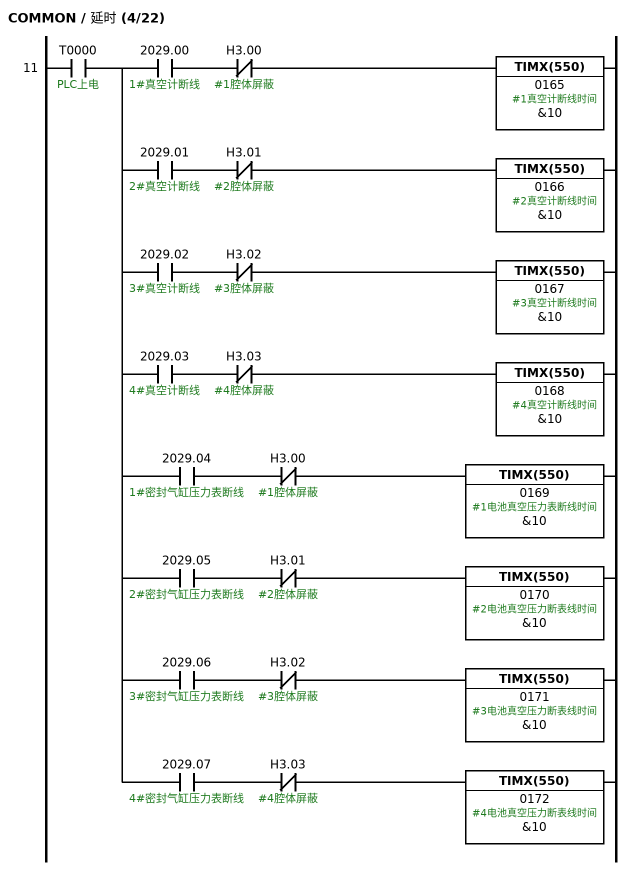
; [picture p384: COMMON / 延时, rungs 11-11]
; rung 11
LD T0000  ; PLC上电
OUT TR0
AND 2029.00  ; 1#真空计断线
ANDNOT H3.00  ; #1腔体屏蔽
TIMX(550) 0165 &10  ; #1真空计断线时间
LD TR0
AND 2029.01  ; 2#真空计断线
ANDNOT H3.01  ; #2腔体屏蔽
TIMX(550) 0166 &10  ; #2真空计断线时间
LD TR0
AND 2029.02  ; 3#真空计断线
ANDNOT H3.02  ; #3腔体屏蔽
TIMX(550) 0167 &10  ; #3真空计断线时间
LD TR0
AND 2029.03  ; 4#真空计断线
ANDNOT H3.03  ; #4腔体屏蔽
TIMX(550) 0168 &10  ; #4真空计断线时间
LD TR0
AND 2029.04  ; 1#密封气缸压力表断线
ANDNOT H3.00  ; #1腔体屏蔽
TIMX(550) 0169 &10  ; #1电池真空压力表断线时间
LD TR0
AND 2029.05  ; 2#密封气缸压力表断线
ANDNOT H3.01  ; #2腔体屏蔽
TIMX(550) 0170 &10  ; #2电池真空压力断表线时间
LD TR0
AND 2029.06  ; 3#密封气缸压力表断线
ANDNOT H3.02  ; #3腔体屏蔽
TIMX(550) 0171 &10  ; #3电池真空压力断表线时间
LD TR0
AND 2029.07  ; 4#密封气缸压力表断线
ANDNOT H3.03  ; #4腔体屏蔽
TIMX(550) 0172 &10  ; #4电池真空压力断表线时间

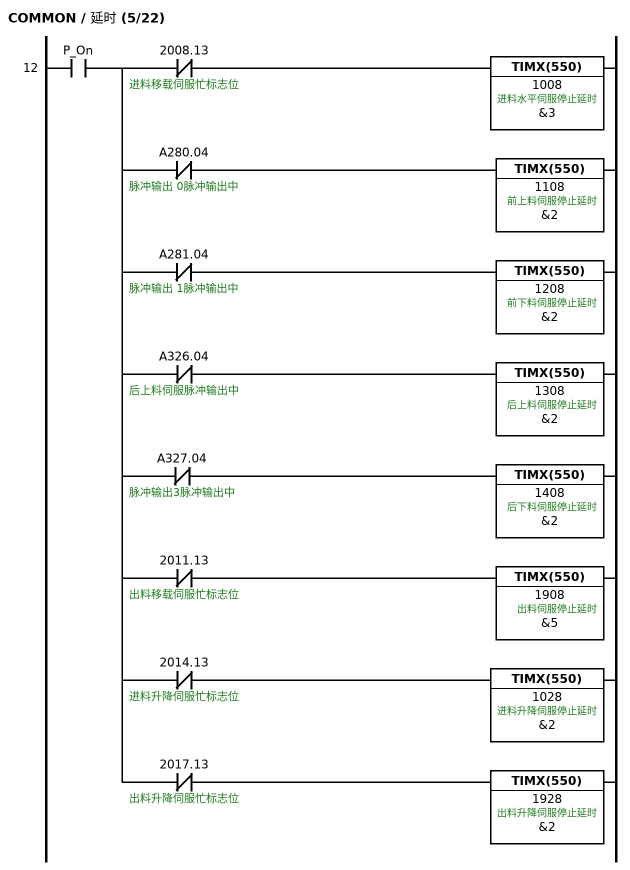
; rung 12
LD P_On
OUT TR0
ANDNOT 2008.13  ; 进料移载伺服忙标志位
TIMX(550) 1008 &3  ; 进料水平伺服停止延时
LD TR0
ANDNOT A280.04  ; 脉冲输出 0脉冲输出中
TIMX(550) 1108 &2  ; 前上料伺服停止延时
LD TR0
ANDNOT A281.04  ; 脉冲输出 1脉冲输出中
TIMX(550) 1208 &2  ; 前下料伺服停止延时
LD TR0
ANDNOT A326.04  ; 后上料伺服脉冲输出中
TIMX(550) 1308 &2  ; 后上料伺服停止延时
LD TR0
ANDNOT A327.04  ; 脉冲输出3脉冲输出中
TIMX(550) 1408 &2  ; 后下料伺服停止延时
LD TR0
ANDNOT 2011.13  ; 出料移载伺服忙标志位
TIMX(550) 1908 &5  ; 出料伺服停止延时
LD TR0
ANDNOT 2014.13  ; 进料升降伺服忙标志位
TIMX(550) 1028 &2  ; 进料升降伺服停止延时
LD TR0
ANDNOT 2017.13  ; 出料升降伺服忙标志位
TIMX(550) 1928 &2  ; 出料升降伺服停止延时

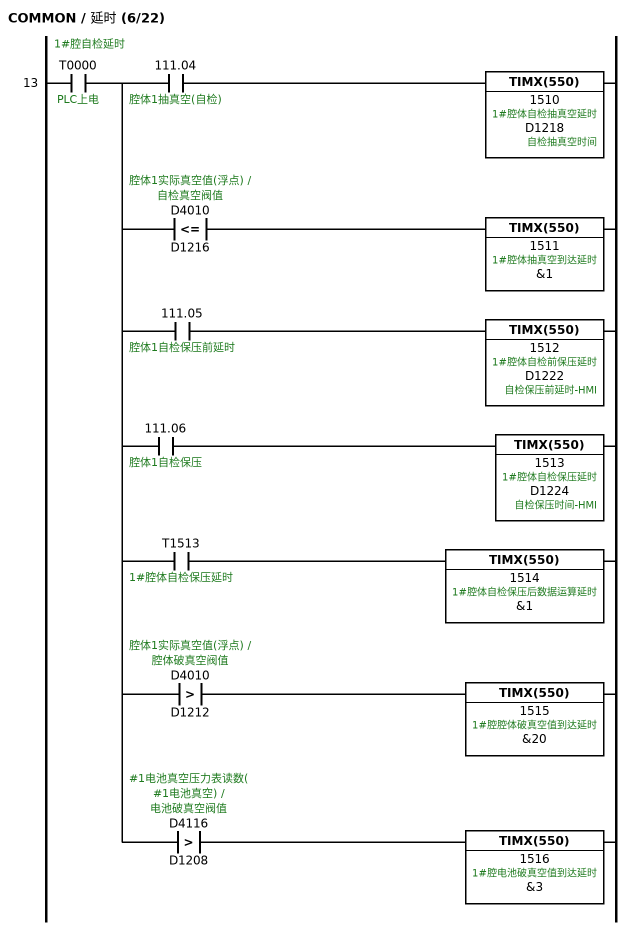
; rung 13: 1#腔自检延时
LD T0000  ; PLC上电
OUT TR0
AND 111.04  ; 腔体1抽真空(自检)
TIMX(550) 1510 D1218  ; 自检抽真空时间, 1#腔体自检抽真空延时
LD TR0
AND<=F(332) D4010 D1216  ; 腔体1实际真空值(浮点), 自检真空阀值
TIMX(550) 1511 &1  ; 1#腔体抽真空到达延时
LD TR0
AND 111.05  ; 腔体1自检保压前延时
TIMX(550) 1512 D1222  ; 自检保压前延时-HMI, 1#腔体自检前保压延时
LD TR0
AND 111.06  ; 腔体1自检保压
TIMX(550) 1513 D1224  ; 自检保压时间-HMI, 1#腔体自检保压延时
LD TR0
AND T1513  ; 1#腔体自检保压延时
TIMX(550) 1514 &1  ; 1#腔体自检保压后数据运算延时
LD TR0
AND>F(333) D4010 D1212  ; 腔体1实际真空值(浮点), 腔体破真空阀值
TIMX(550) 1515 &20  ; 1#腔腔体破真空值到达延时
LD TR0
AND>F(333) D4116 D1208  ; #1电池真空压力表读数(#1电池真空), 电池破真空阀值
TIMX(550) 1516 &3  ; 1#腔电池破真空值到达延时

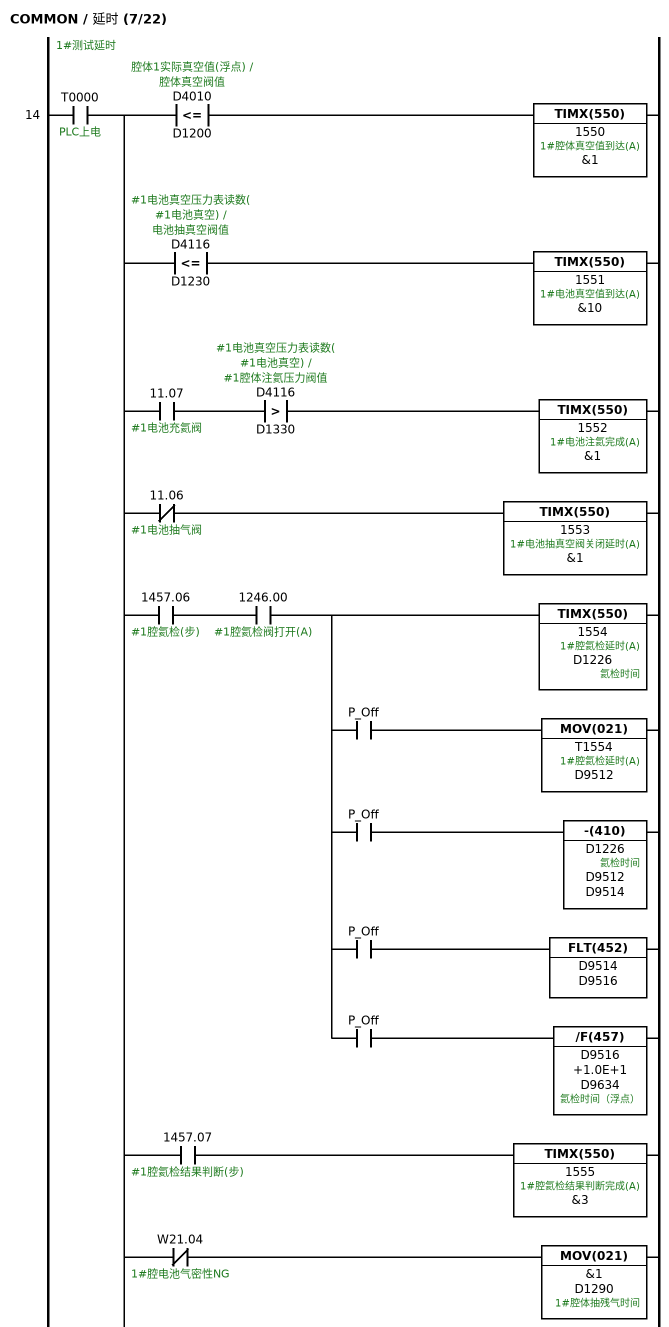

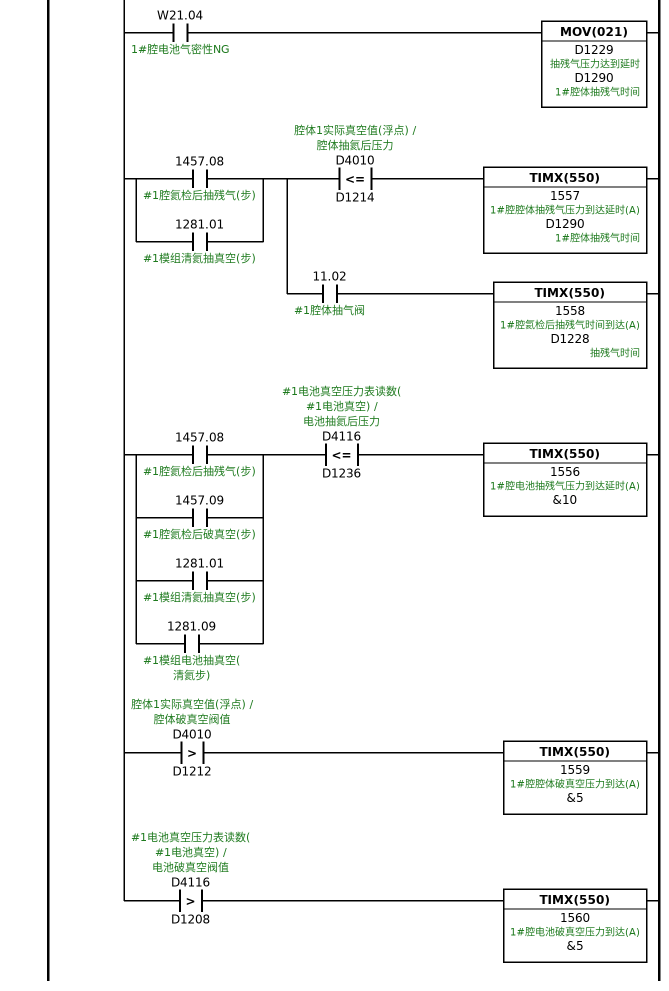
; rung 14: 1#测试延时
LD T0000  ; PLC上电
OUT TR0
AND<=F(332) D4010 D1200  ; 腔体1实际真空值(浮点), 腔体真空阀值
TIMX(550) 1550 &1  ; 1#腔体真空值到达(A)
LD TR0
AND<=F(332) D4116 D1230  ; #1电池真空压力表读数(#1电池真空), 电池抽真空阀值
TIMX(550) 1551 &10  ; 1#电池真空值到达(A)
LD TR0
AND 11.07  ; #1电池充氦阀
AND>F(333) D4116 D1330  ; #1电池真空压力表读数(#1电池真空), #1腔体注氦压力阀值
TIMX(550) 1552 &1  ; 1#电池注氦完成(A)
LD TR0
ANDNOT 11.06  ; #1电池抽气阀
TIMX(550) 1553 &1  ; 1#电池抽真空阀关闭延时(A)
LD TR0
AND 1457.06  ; #1腔氦检(步)
AND 1246.00  ; #1腔氦检阀打开(A)
OUT TR1
TIMX(550) 1554 D1226  ; 氦检时间, 1#腔氦检延时(A)
AND P_Off
MOV(021) T1554 D9512  ; 1#腔氦检延时(A)
LD TR1
AND P_Off
-(410) D1226 D9512 D9514  ; 氦检时间
LD TR1
AND P_Off
FLT(452) D9514 D9516
LD TR1
AND P_Off
/F(457) D9516 +1.0E+1 D9634  ; 氦检时间（浮点）
LD TR0
AND 1457.07  ; #1腔氦检结果判断(步)
TIMX(550) 1555 &3  ; 1#腔氦检结果判断完成(A)
LD TR0
ANDNOT W21.04  ; 1#腔电池气密性NG
MOV(021) &1 D1290  ; 1#腔体抽残气时间
LD TR0
AND W21.04  ; 1#腔电池气密性NG
MOV(021) D1229 D1290  ; 抽残气压力达到延时, 1#腔体抽残气时间
LD TR0
LD 1457.08  ; #1腔氦检后抽残气(步)
OR 1281.01  ; #1模组清氦抽真空(步)
ANDLD
OUT TR1
AND<=F(332) D4010 D1214  ; 腔体1实际真空值(浮点), 腔体抽氦后压力
TIMX(550) 1557 D1290  ; 1#腔体抽残气时间, 1#腔腔体抽残气压力到达延时(A)
LD TR1
AND 11.02  ; #1腔体抽气阀
TIMX(550) 1558 D1228  ; 抽残气时间, 1#腔氦检后抽残气时间到达(A)
LD TR0
LD 1457.08  ; #1腔氦检后抽残气(步)
OR 1457.09  ; #1腔氦检后破真空(步)
OR 1281.01  ; #1模组清氦抽真空(步)
OR 1281.09  ; #1模组电池抽真空(清氦步)
ANDLD
AND<=F(332) D4116 D1236  ; #1电池真空压力表读数(#1电池真空), 电池抽氦后压力
TIMX(550) 1556 &10  ; 1#腔电池抽残气压力到达延时(A)
LD TR0
AND>F(333) D4010 D1212  ; 腔体1实际真空值(浮点), 腔体破真空阀值
TIMX(550) 1559 &5  ; 1#腔腔体破真空压力到达(A)
LD TR0
AND>F(333) D4116 D1208  ; #1电池真空压力表读数(#1电池真空), 电池破真空阀值
TIMX(550) 1560 &5  ; 1#腔电池破真空压力到达(A)

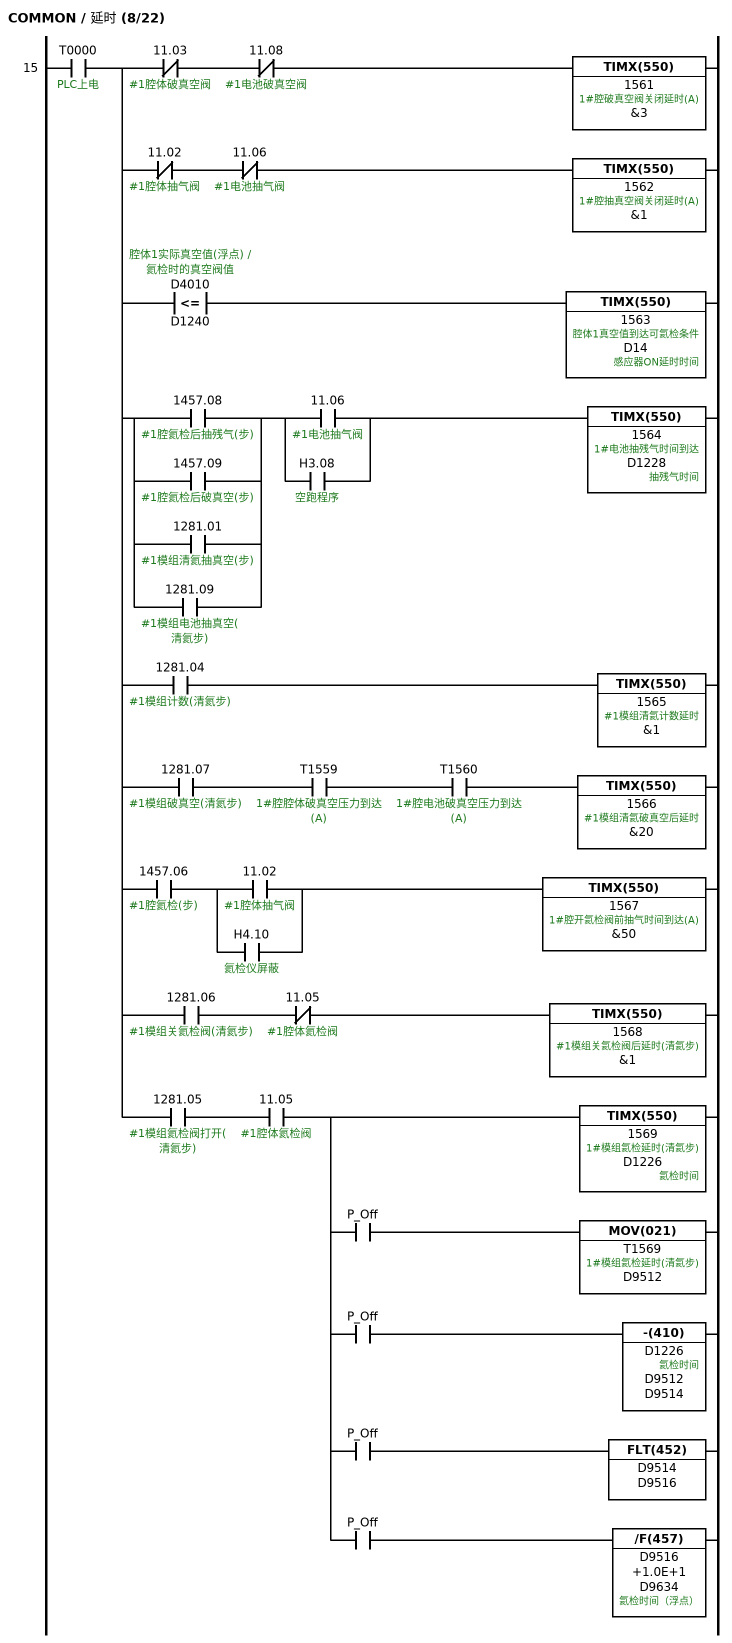
; rung 15
LD T0000  ; PLC上电
OUT TR0
ANDNOT 11.03  ; #1腔体破真空阀
ANDNOT 11.08  ; #1电池破真空阀
TIMX(550) 1561 &3  ; 1#腔破真空阀关闭延时(A)
LD TR0
ANDNOT 11.02  ; #1腔体抽气阀
ANDNOT 11.06  ; #1电池抽气阀
TIMX(550) 1562 &1  ; 1#腔抽真空阀关闭延时(A)
LD TR0
AND<=F(332) D4010 D1240  ; 腔体1实际真空值(浮点), 氦检时的真空阀值
TIMX(550) 1563 D14  ; 感应器ON延时时间, 腔体1真空值到达可氦检条件
LD TR0
LD 1457.08  ; #1腔氦检后抽残气(步)
OR 1457.09  ; #1腔氦检后破真空(步)
OR 1281.01  ; #1模组清氦抽真空(步)
OR 1281.09  ; #1模组电池抽真空(清氦步)
ANDLD
LD 11.06  ; #1电池抽气阀
OR H3.08  ; 空跑程序
ANDLD
TIMX(550) 1564 D1228  ; 抽残气时间, 1#电池抽残气时间到达
LD TR0
AND 1281.04  ; #1模组计数(清氦步)
TIMX(550) 1565 &1  ; #1模组清氦计数延时
LD TR0
AND 1281.07  ; #1模组破真空(清氦步)
AND T1559  ; 1#腔腔体破真空压力到达(A)
AND T1560  ; 1#腔电池破真空压力到达(A)
TIMX(550) 1566 &20  ; #1模组清氦破真空后延时
LD TR0
AND 1457.06  ; #1腔氦检(步)
LD 11.02  ; #1腔体抽气阀
OR H4.10  ; 氦检仪屏蔽
ANDLD
TIMX(550) 1567 &50  ; 1#腔开氦检阀前抽气时间到达(A)
LD TR0
AND 1281.06  ; #1模组关氦检阀(清氦步)
ANDNOT 11.05  ; #1腔体氦检阀
TIMX(550) 1568 &1  ; #1模组关氦检阀后延时(清氦步)
LD TR0
AND 1281.05  ; #1模组氦检阀打开(清氦步)
AND 11.05  ; #1腔体氦检阀
OUT TR0
TIMX(550) 1569 D1226  ; 氦检时间, 1#模组氦检延时(清氦步)
AND P_Off
MOV(021) T1569 D9512  ; 1#模组氦检延时(清氦步)
LD TR0
AND P_Off
-(410) D1226 D9512 D9514  ; 氦检时间
LD TR0
AND P_Off
FLT(452) D9514 D9516
LD TR0
AND P_Off
/F(457) D9516 +1.0E+1 D9634  ; 氦检时间（浮点）

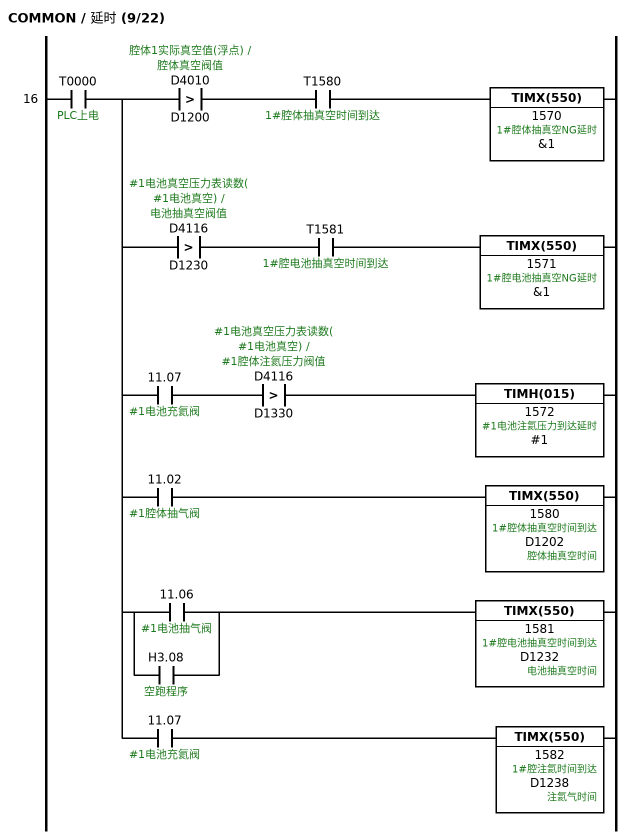
; rung 16
LD T0000  ; PLC上电
OUT TR0
AND>F(333) D4010 D1200  ; 腔体1实际真空值(浮点), 腔体真空阀值
AND T1580  ; 1#腔体抽真空时间到达
TIMX(550) 1570 &1  ; 1#腔体抽真空NG延时
LD TR0
AND>F(333) D4116 D1230  ; #1电池真空压力表读数(#1电池真空), 电池抽真空阀值
AND T1581  ; 1#腔电池抽真空时间到达
TIMX(550) 1571 &1  ; 1#腔电池抽真空NG延时
LD TR0
AND 11.07  ; #1电池充氦阀
AND>F(333) D4116 D1330  ; #1电池真空压力表读数(#1电池真空), #1腔体注氦压力阀值
TIMH(015) 1572 #1  ; #1电池注氦压力到达延时
LD TR0
AND 11.02  ; #1腔体抽气阀
TIMX(550) 1580 D1202  ; 腔体抽真空时间, 1#腔体抽真空时间到达
LD TR0
LD 11.06  ; #1电池抽气阀
OR H3.08  ; 空跑程序
ANDLD
TIMX(550) 1581 D1232  ; 电池抽真空时间, 1#腔电池抽真空时间到达
LD TR0
AND 11.07  ; #1电池充氦阀
TIMX(550) 1582 D1238  ; 注氦气时间, 1#腔注氦时间到达

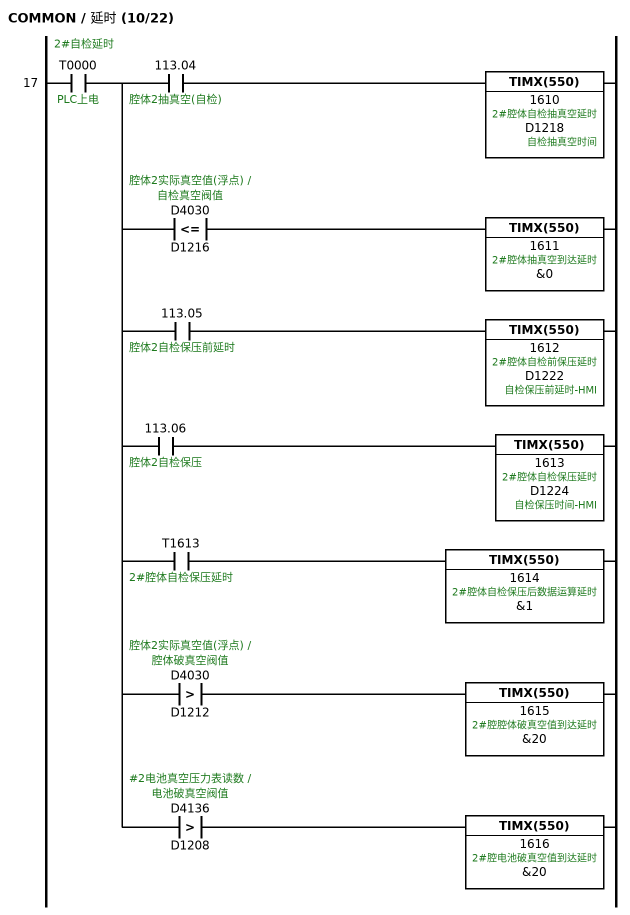
; rung 17: 2#自检延时
LD T0000  ; PLC上电
OUT TR0
AND 113.04  ; 腔体2抽真空(自检)
TIMX(550) 1610 D1218  ; 自检抽真空时间, 2#腔体自检抽真空延时
LD TR0
AND<=F(332) D4030 D1216  ; 腔体2实际真空值(浮点), 自检真空阀值
TIMX(550) 1611 &0  ; 2#腔体抽真空到达延时
LD TR0
AND 113.05  ; 腔体2自检保压前延时
TIMX(550) 1612 D1222  ; 自检保压前延时-HMI, 2#腔体自检前保压延时
LD TR0
AND 113.06  ; 腔体2自检保压
TIMX(550) 1613 D1224  ; 自检保压时间-HMI, 2#腔体自检保压延时
LD TR0
AND T1613  ; 2#腔体自检保压延时
TIMX(550) 1614 &1  ; 2#腔体自检保压后数据运算延时
LD TR0
AND>F(333) D4030 D1212  ; 腔体2实际真空值(浮点), 腔体破真空阀值
TIMX(550) 1615 &20  ; 2#腔腔体破真空值到达延时
LD TR0
AND>F(333) D4136 D1208  ; #2电池真空压力表读数, 电池破真空阀值
TIMX(550) 1616 &20  ; 2#腔电池破真空值到达延时

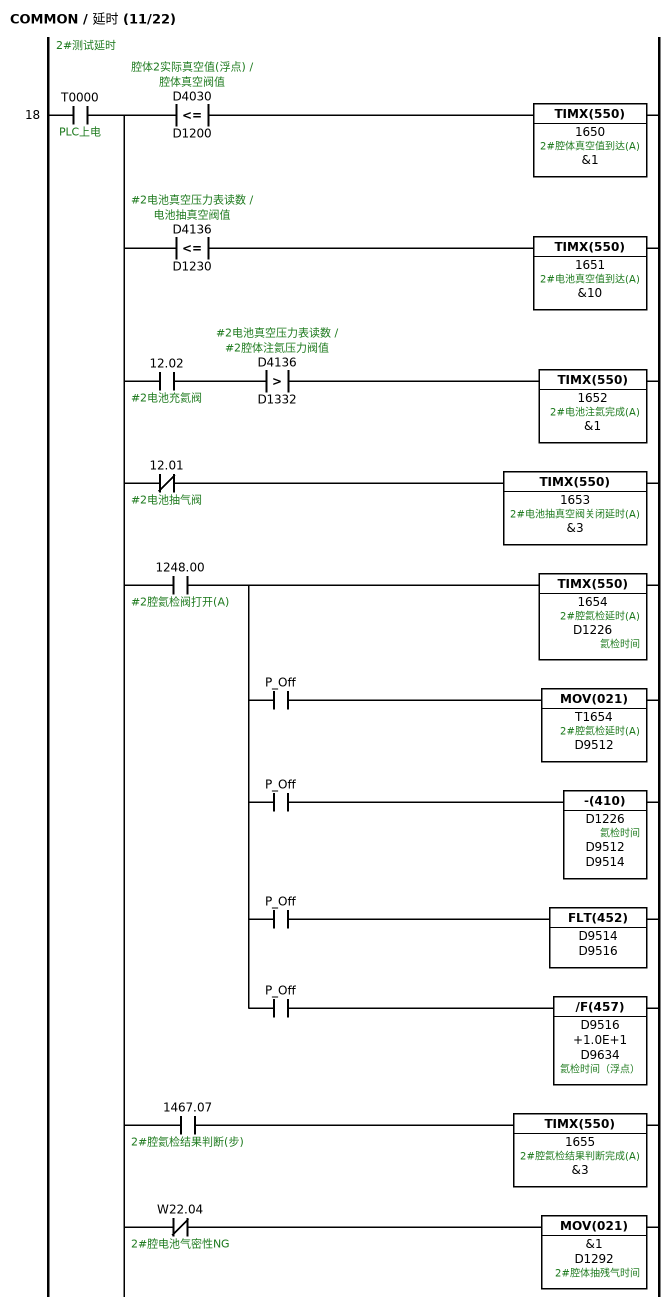

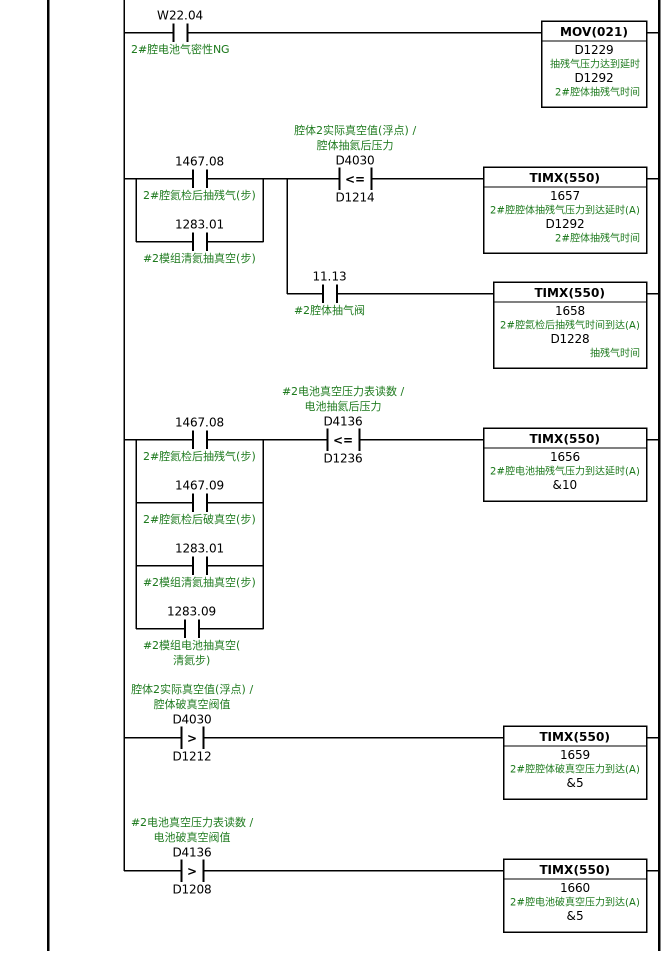
; rung 18: 2#测试延时
LD T0000  ; PLC上电
OUT TR0
AND<=F(332) D4030 D1200  ; 腔体2实际真空值(浮点), 腔体真空阀值
TIMX(550) 1650 &1  ; 2#腔体真空值到达(A)
LD TR0
AND<=F(332) D4136 D1230  ; #2电池真空压力表读数, 电池抽真空阀值
TIMX(550) 1651 &10  ; 2#电池真空值到达(A)
LD TR0
AND 12.02  ; #2电池充氦阀
AND>F(333) D4136 D1332  ; #2电池真空压力表读数, #2腔体注氦压力阀值
TIMX(550) 1652 &1  ; 2#电池注氦完成(A)
LD TR0
ANDNOT 12.01  ; #2电池抽气阀
TIMX(550) 1653 &3  ; 2#电池抽真空阀关闭延时(A)
LD TR0
AND 1248.00  ; #2腔氦检阀打开(A)
OUT TR1
TIMX(550) 1654 D1226  ; 氦检时间, 2#腔氦检延时(A)
AND P_Off
MOV(021) T1654 D9512  ; 2#腔氦检延时(A)
LD TR1
AND P_Off
-(410) D1226 D9512 D9514  ; 氦检时间
LD TR1
AND P_Off
FLT(452) D9514 D9516
LD TR1
AND P_Off
/F(457) D9516 +1.0E+1 D9634  ; 氦检时间（浮点）
LD TR0
AND 1467.07  ; 2#腔氦检结果判断(步)
TIMX(550) 1655 &3  ; 2#腔氦检结果判断完成(A)
LD TR0
ANDNOT W22.04  ; 2#腔电池气密性NG
MOV(021) &1 D1292  ; 2#腔体抽残气时间
LD TR0
AND W22.04  ; 2#腔电池气密性NG
MOV(021) D1229 D1292  ; 抽残气压力达到延时, 2#腔体抽残气时间
LD TR0
LD 1467.08  ; 2#腔氦检后抽残气(步)
OR 1283.01  ; #2模组清氦抽真空(步)
ANDLD
OUT TR1
AND<=F(332) D4030 D1214  ; 腔体2实际真空值(浮点), 腔体抽氦后压力
TIMX(550) 1657 D1292  ; 2#腔体抽残气时间, 2#腔腔体抽残气压力到达延时(A)
LD TR1
AND 11.13  ; #2腔体抽气阀
TIMX(550) 1658 D1228  ; 抽残气时间, 2#腔氦检后抽残气时间到达(A)
LD TR0
LD 1467.08  ; 2#腔氦检后抽残气(步)
OR 1467.09  ; 2#腔氦检后破真空(步)
OR 1283.01  ; #2模组清氦抽真空(步)
OR 1283.09  ; #2模组电池抽真空(清氦步)
ANDLD
AND<=F(332) D4136 D1236  ; #2电池真空压力表读数, 电池抽氦后压力
TIMX(550) 1656 &10  ; 2#腔电池抽残气压力到达延时(A)
LD TR0
AND>F(333) D4030 D1212  ; 腔体2实际真空值(浮点), 腔体破真空阀值
TIMX(550) 1659 &5  ; 2#腔腔体破真空压力到达(A)
LD TR0
AND>F(333) D4136 D1208  ; #2电池真空压力表读数, 电池破真空阀值
TIMX(550) 1660 &5  ; 2#腔电池破真空压力到达(A)

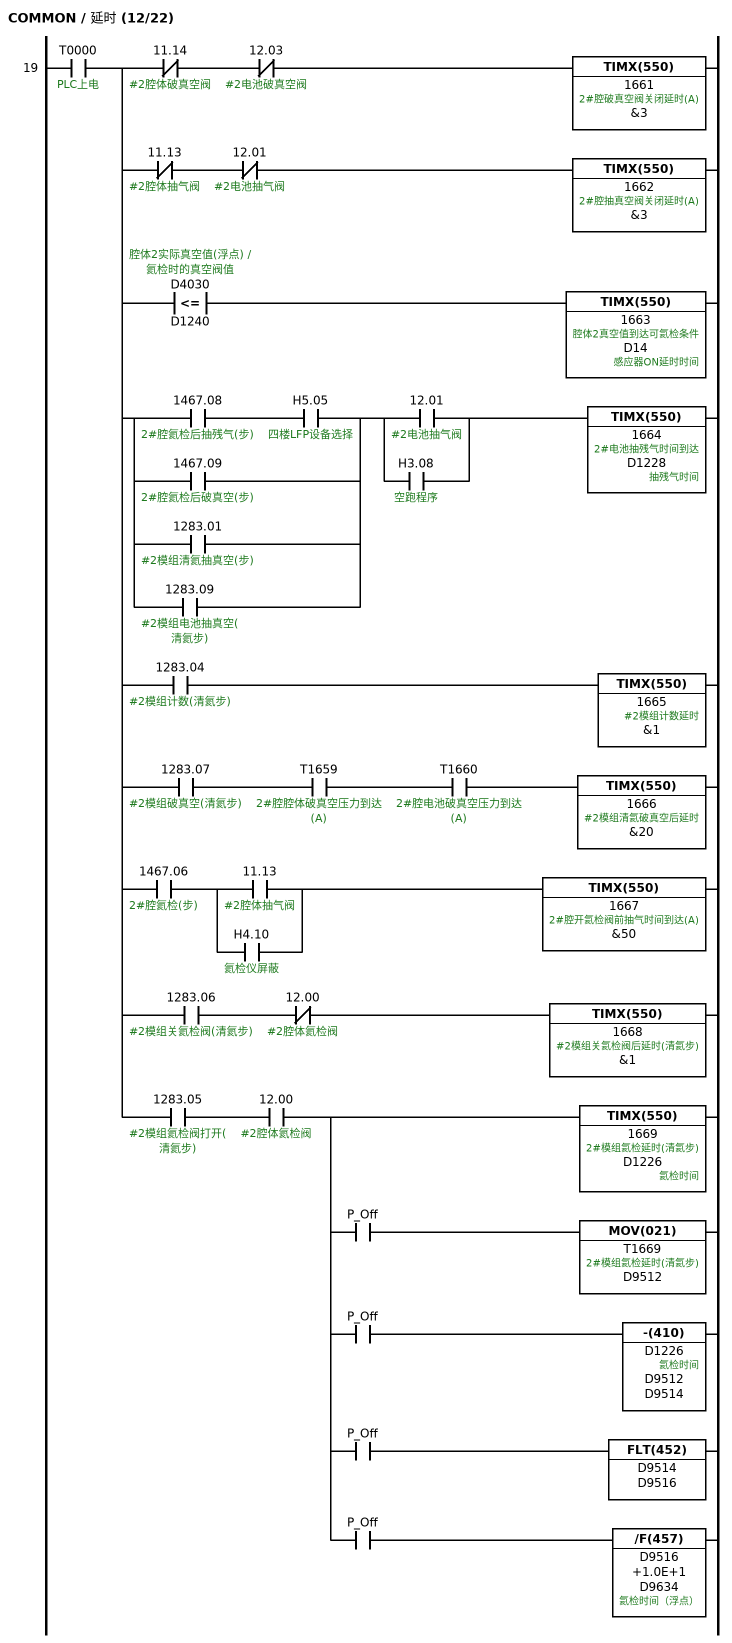
; rung 19
LD T0000  ; PLC上电
OUT TR0
ANDNOT 11.14  ; #2腔体破真空阀
ANDNOT 12.03  ; #2电池破真空阀
TIMX(550) 1661 &3  ; 2#腔破真空阀关闭延时(A)
LD TR0
ANDNOT 11.13  ; #2腔体抽气阀
ANDNOT 12.01  ; #2电池抽气阀
TIMX(550) 1662 &3  ; 2#腔抽真空阀关闭延时(A)
LD TR0
AND<=F(332) D4030 D1240  ; 腔体2实际真空值(浮点), 氦检时的真空阀值
TIMX(550) 1663 D14  ; 感应器ON延时时间, 腔体2真空值到达可氦检条件
LD TR0
LD 1467.08  ; 2#腔氦检后抽残气(步)
AND H5.05  ; 四楼LFP设备选择
OR 1467.09  ; 2#腔氦检后破真空(步)
OR 1283.01  ; #2模组清氦抽真空(步)
OR 1283.09  ; #2模组电池抽真空(清氦步)
ANDLD
LD 12.01  ; #2电池抽气阀
OR H3.08  ; 空跑程序
ANDLD
TIMX(550) 1664 D1228  ; 抽残气时间, 2#电池抽残气时间到达
LD TR0
AND 1283.04  ; #2模组计数(清氦步)
TIMX(550) 1665 &1  ; #2模组计数延时
LD TR0
AND 1283.07  ; #2模组破真空(清氦步)
AND T1659  ; 2#腔腔体破真空压力到达(A)
AND T1660  ; 2#腔电池破真空压力到达(A)
TIMX(550) 1666 &20  ; #2模组清氦破真空后延时
LD TR0
AND 1467.06  ; 2#腔氦检(步)
LD 11.13  ; #2腔体抽气阀
OR H4.10  ; 氦检仪屏蔽
ANDLD
TIMX(550) 1667 &50  ; 2#腔开氦检阀前抽气时间到达(A)
LD TR0
AND 1283.06  ; #2模组关氦检阀(清氦步)
ANDNOT 12.00  ; #2腔体氦检阀
TIMX(550) 1668 &1  ; #2模组关氦检阀后延时(清氦步)
LD TR0
AND 1283.05  ; #2模组氦检阀打开(清氦步)
AND 12.00  ; #2腔体氦检阀
OUT TR0
TIMX(550) 1669 D1226  ; 氦检时间, 2#模组氦检延时(清氦步)
AND P_Off
MOV(021) T1669 D9512  ; 2#模组氦检延时(清氦步)
LD TR0
AND P_Off
-(410) D1226 D9512 D9514  ; 氦检时间
LD TR0
AND P_Off
FLT(452) D9514 D9516
LD TR0
AND P_Off
/F(457) D9516 +1.0E+1 D9634  ; 氦检时间（浮点）

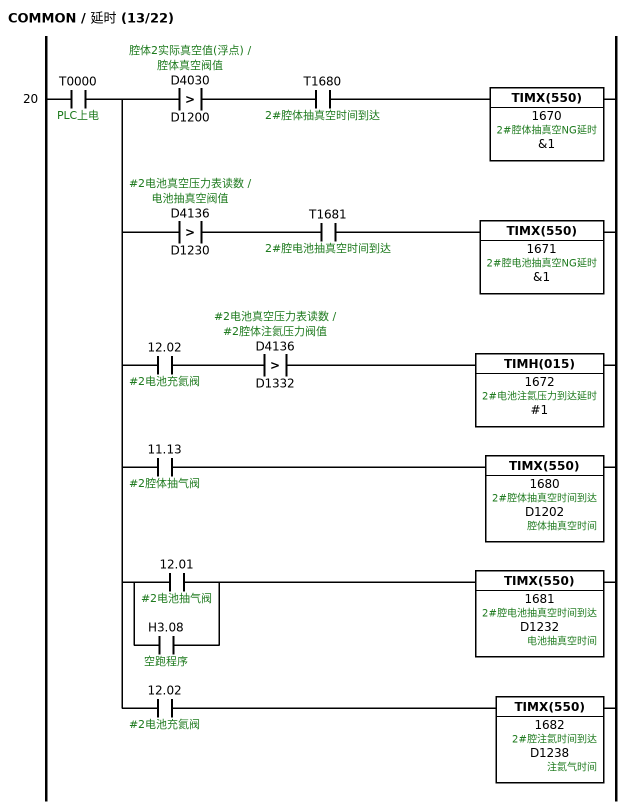
; rung 20
LD T0000  ; PLC上电
OUT TR0
AND>F(333) D4030 D1200  ; 腔体2实际真空值(浮点), 腔体真空阀值
AND T1680  ; 2#腔体抽真空时间到达
TIMX(550) 1670 &1  ; 2#腔体抽真空NG延时
LD TR0
AND>F(333) D4136 D1230  ; #2电池真空压力表读数, 电池抽真空阀值
AND T1681  ; 2#腔电池抽真空时间到达
TIMX(550) 1671 &1  ; 2#腔电池抽真空NG延时
LD TR0
AND 12.02  ; #2电池充氦阀
AND>F(333) D4136 D1332  ; #2电池真空压力表读数, #2腔体注氦压力阀值
TIMH(015) 1672 #1  ; 2#电池注氦压力到达延时
LD TR0
AND 11.13  ; #2腔体抽气阀
TIMX(550) 1680 D1202  ; 腔体抽真空时间, 2#腔体抽真空时间到达
LD TR0
LD 12.01  ; #2电池抽气阀
OR H3.08  ; 空跑程序
ANDLD
TIMX(550) 1681 D1232  ; 电池抽真空时间, 2#腔电池抽真空时间到达
LD TR0
AND 12.02  ; #2电池充氦阀
TIMX(550) 1682 D1238  ; 注氦气时间, 2#腔注氦时间到达

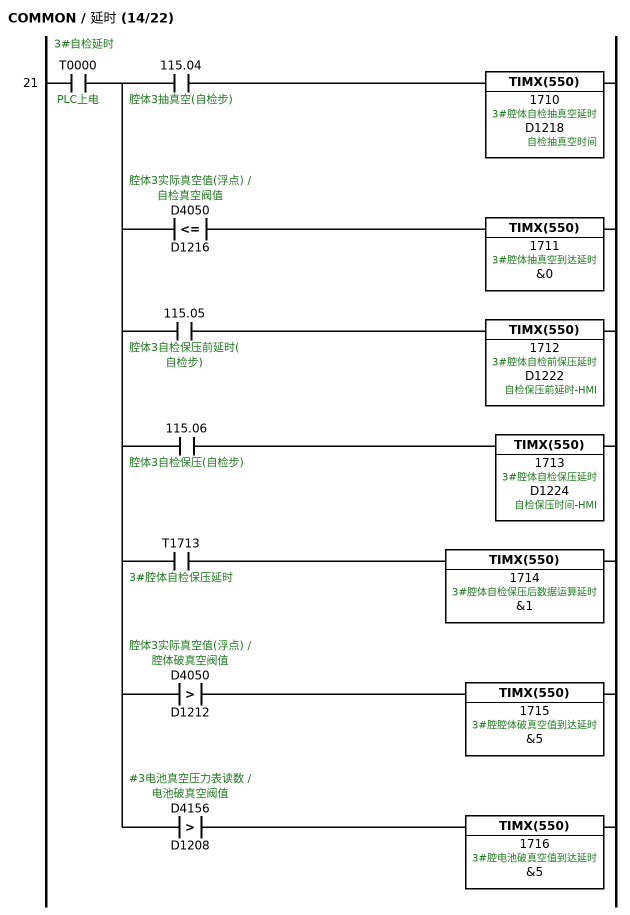
; rung 21: 3#自检延时
LD T0000  ; PLC上电
OUT TR0
AND 115.04  ; 腔体3抽真空(自检步)
TIMX(550) 1710 D1218  ; 自检抽真空时间, 3#腔体自检抽真空延时
LD TR0
AND<=F(332) D4050 D1216  ; 腔体3实际真空值(浮点), 自检真空阀值
TIMX(550) 1711 &0  ; 3#腔体抽真空到达延时
LD TR0
AND 115.05  ; 腔体3自检保压前延时(自检步)
TIMX(550) 1712 D1222  ; 自检保压前延时-HMI, 3#腔体自检前保压延时
LD TR0
AND 115.06  ; 腔体3自检保压(自检步)
TIMX(550) 1713 D1224  ; 自检保压时间-HMI, 3#腔体自检保压延时
LD TR0
AND T1713  ; 3#腔体自检保压延时
TIMX(550) 1714 &1  ; 3#腔体自检保压后数据运算延时
LD TR0
AND>F(333) D4050 D1212  ; 腔体3实际真空值(浮点), 腔体破真空阀值
TIMX(550) 1715 &5  ; 3#腔腔体破真空值到达延时
LD TR0
AND>F(333) D4156 D1208  ; #3电池真空压力表读数, 电池破真空阀值
TIMX(550) 1716 &5  ; 3#腔电池破真空值到达延时

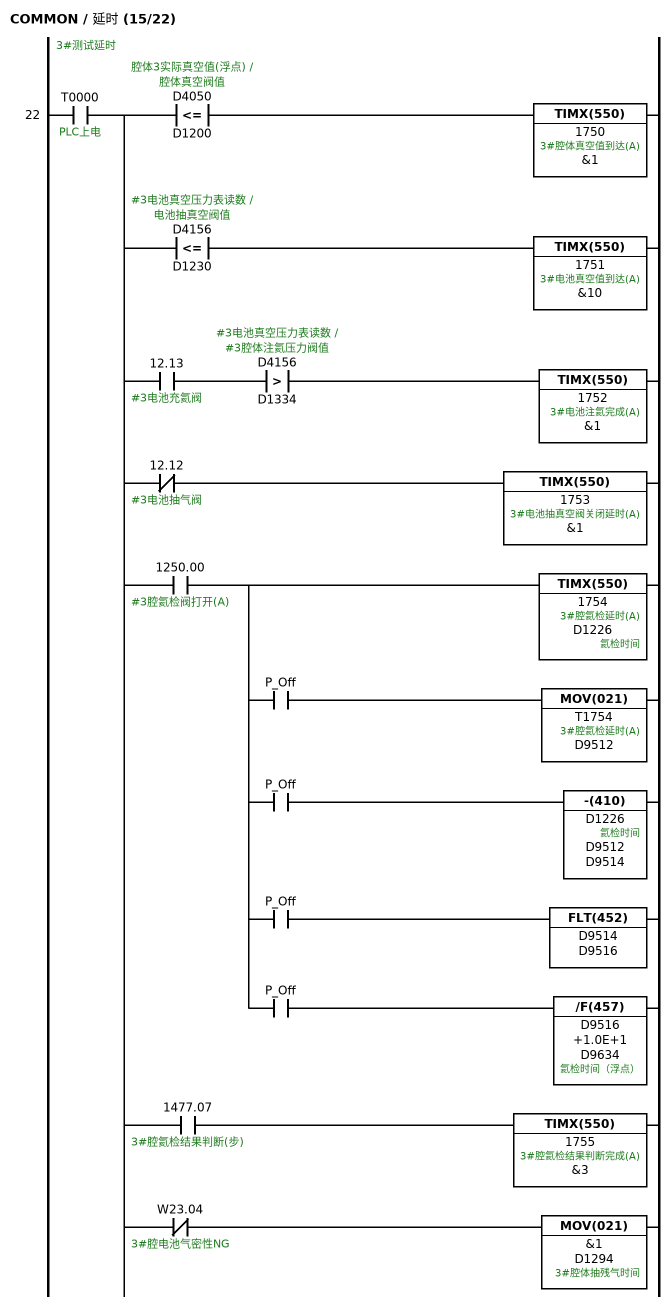

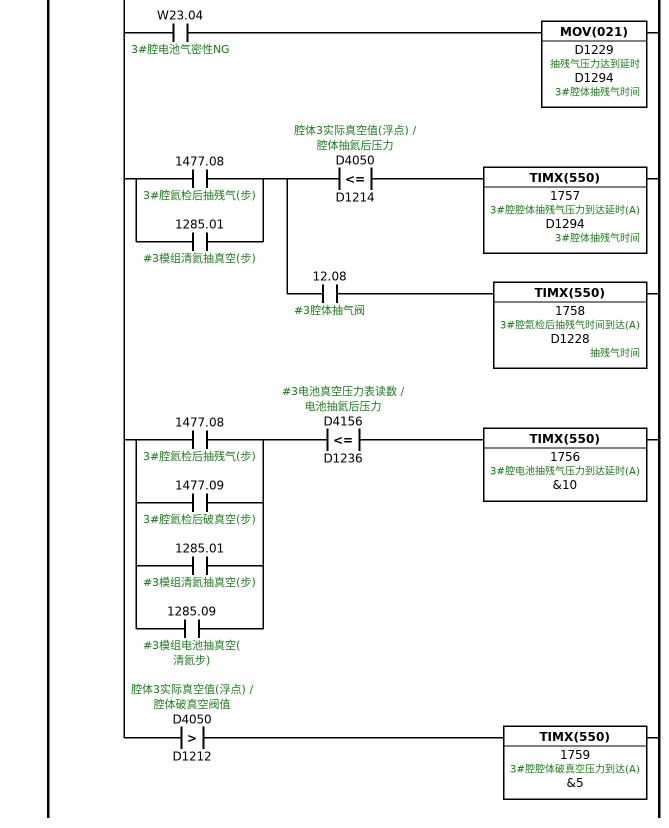
; rung 22: 3#测试延时
LD T0000  ; PLC上电
OUT TR0
AND<=F(332) D4050 D1200  ; 腔体3实际真空值(浮点), 腔体真空阀值
TIMX(550) 1750 &1  ; 3#腔体真空值到达(A)
LD TR0
AND<=F(332) D4156 D1230  ; #3电池真空压力表读数, 电池抽真空阀值
TIMX(550) 1751 &10  ; 3#电池真空值到达(A)
LD TR0
AND 12.13  ; #3电池充氦阀
AND>F(333) D4156 D1334  ; #3电池真空压力表读数, #3腔体注氦压力阀值
TIMX(550) 1752 &1  ; 3#电池注氦完成(A)
LD TR0
ANDNOT 12.12  ; #3电池抽气阀
TIMX(550) 1753 &1  ; 3#电池抽真空阀关闭延时(A)
LD TR0
AND 1250.00  ; #3腔氦检阀打开(A)
OUT TR1
TIMX(550) 1754 D1226  ; 氦检时间, 3#腔氦检延时(A)
AND P_Off
MOV(021) T1754 D9512  ; 3#腔氦检延时(A)
LD TR1
AND P_Off
-(410) D1226 D9512 D9514  ; 氦检时间
LD TR1
AND P_Off
FLT(452) D9514 D9516
LD TR1
AND P_Off
/F(457) D9516 +1.0E+1 D9634  ; 氦检时间（浮点）
LD TR0
AND 1477.07  ; 3#腔氦检结果判断(步)
TIMX(550) 1755 &3  ; 3#腔氦检结果判断完成(A)
LD TR0
ANDNOT W23.04  ; 3#腔电池气密性NG
MOV(021) &1 D1294  ; 3#腔体抽残气时间
LD TR0
AND W23.04  ; 3#腔电池气密性NG
MOV(021) D1229 D1294  ; 抽残气压力达到延时, 3#腔体抽残气时间
LD TR0
LD 1477.08  ; 3#腔氦检后抽残气(步)
OR 1285.01  ; #3模组清氦抽真空(步)
ANDLD
OUT TR1
AND<=F(332) D4050 D1214  ; 腔体3实际真空值(浮点), 腔体抽氦后压力
TIMX(550) 1757 D1294  ; 3#腔体抽残气时间, 3#腔腔体抽残气压力到达延时(A)
LD TR1
AND 12.08  ; #3腔体抽气阀
TIMX(550) 1758 D1228  ; 抽残气时间, 3#腔氦检后抽残气时间到达(A)
LD TR0
LD 1477.08  ; 3#腔氦检后抽残气(步)
OR 1477.09  ; 3#腔氦检后破真空(步)
OR 1285.01  ; #3模组清氦抽真空(步)
OR 1285.09  ; #3模组电池抽真空(清氦步)
ANDLD
AND<=F(332) D4156 D1236  ; #3电池真空压力表读数, 电池抽氦后压力
TIMX(550) 1756 &10  ; 3#腔电池抽残气压力到达延时(A)
LD TR0
AND>F(333) D4050 D1212  ; 腔体3实际真空值(浮点), 腔体破真空阀值
TIMX(550) 1759 &5  ; 3#腔腔体破真空压力到达(A)

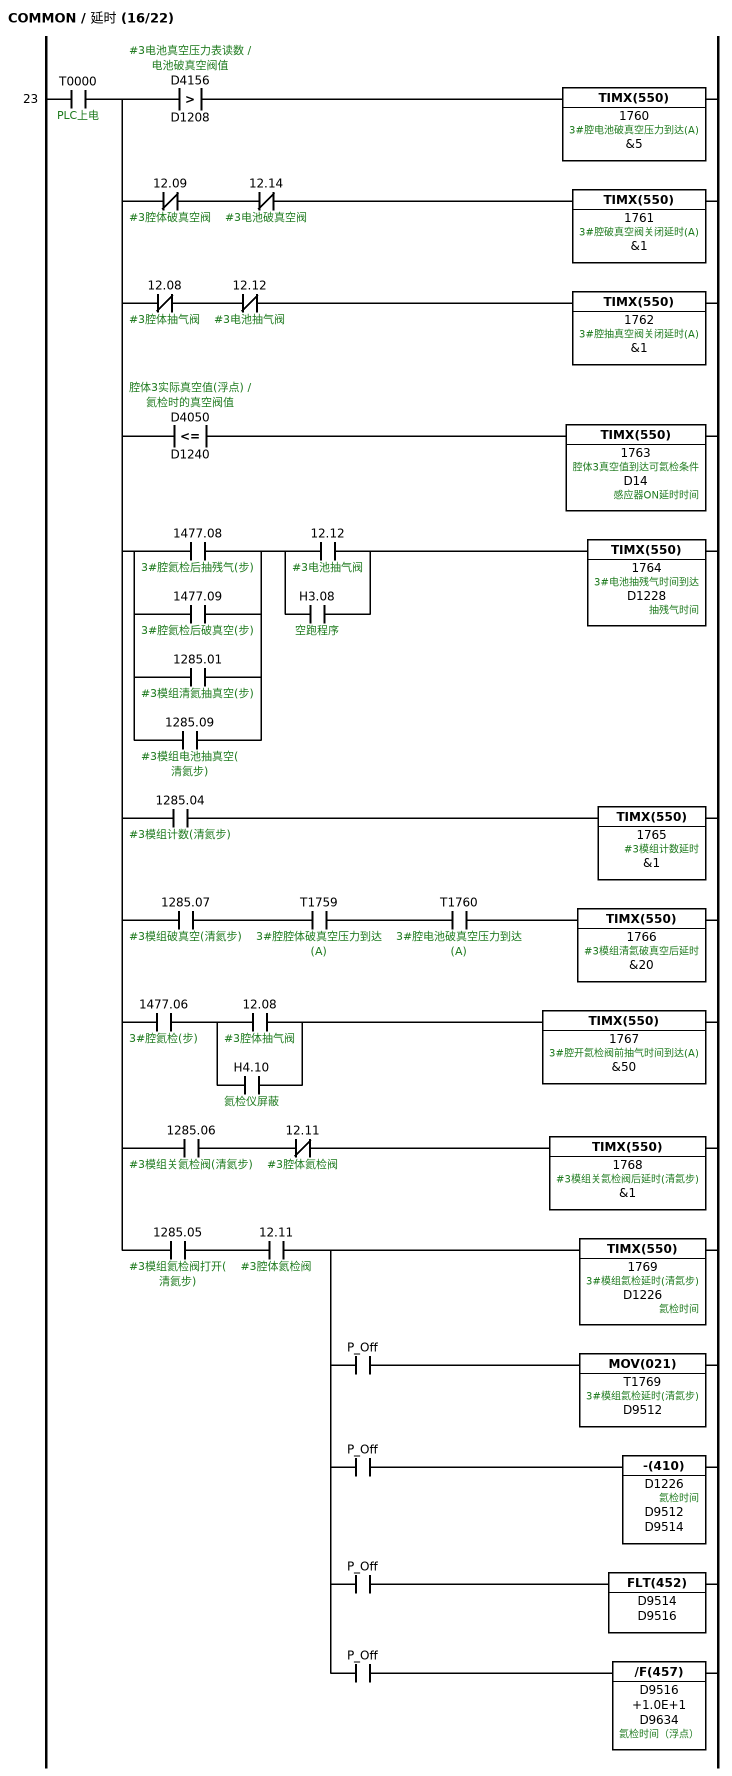
; rung 23
LD T0000  ; PLC上电
OUT TR0
AND>F(333) D4156 D1208  ; #3电池真空压力表读数, 电池破真空阀值
TIMX(550) 1760 &5  ; 3#腔电池破真空压力到达(A)
LD TR0
ANDNOT 12.09  ; #3腔体破真空阀
ANDNOT 12.14  ; #3电池破真空阀
TIMX(550) 1761 &1  ; 3#腔破真空阀关闭延时(A)
LD TR0
ANDNOT 12.08  ; #3腔体抽气阀
ANDNOT 12.12  ; #3电池抽气阀
TIMX(550) 1762 &1  ; 3#腔抽真空阀关闭延时(A)
LD TR0
AND<=F(332) D4050 D1240  ; 腔体3实际真空值(浮点), 氦检时的真空阀值
TIMX(550) 1763 D14  ; 感应器ON延时时间, 腔体3真空值到达可氦检条件
LD TR0
LD 1477.08  ; 3#腔氦检后抽残气(步)
OR 1477.09  ; 3#腔氦检后破真空(步)
OR 1285.01  ; #3模组清氦抽真空(步)
OR 1285.09  ; #3模组电池抽真空(清氦步)
ANDLD
LD 12.12  ; #3电池抽气阀
OR H3.08  ; 空跑程序
ANDLD
TIMX(550) 1764 D1228  ; 抽残气时间, 3#电池抽残气时间到达
LD TR0
AND 1285.04  ; #3模组计数(清氦步)
TIMX(550) 1765 &1  ; #3模组计数延时
LD TR0
AND 1285.07  ; #3模组破真空(清氦步)
AND T1759  ; 3#腔腔体破真空压力到达(A)
AND T1760  ; 3#腔电池破真空压力到达(A)
TIMX(550) 1766 &20  ; #3模组清氦破真空后延时
LD TR0
AND 1477.06  ; 3#腔氦检(步)
LD 12.08  ; #3腔体抽气阀
OR H4.10  ; 氦检仪屏蔽
ANDLD
TIMX(550) 1767 &50  ; 3#腔开氦检阀前抽气时间到达(A)
LD TR0
AND 1285.06  ; #3模组关氦检阀(清氦步)
ANDNOT 12.11  ; #3腔体氦检阀
TIMX(550) 1768 &1  ; #3模组关氦检阀后延时(清氦步)
LD TR0
AND 1285.05  ; #3模组氦检阀打开(清氦步)
AND 12.11  ; #3腔体氦检阀
OUT TR0
TIMX(550) 1769 D1226  ; 氦检时间, 3#模组氦检延时(清氦步)
AND P_Off
MOV(021) T1769 D9512  ; 3#模组氦检延时(清氦步)
LD TR0
AND P_Off
-(410) D1226 D9512 D9514  ; 氦检时间
LD TR0
AND P_Off
FLT(452) D9514 D9516
LD TR0
AND P_Off
/F(457) D9516 +1.0E+1 D9634  ; 氦检时间（浮点）

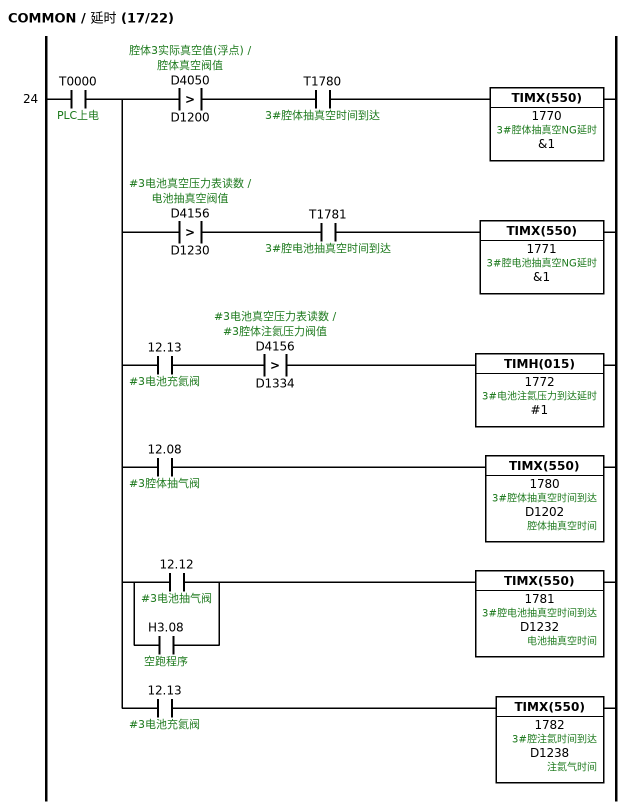
; rung 24
LD T0000  ; PLC上电
OUT TR0
AND>F(333) D4050 D1200  ; 腔体3实际真空值(浮点), 腔体真空阀值
AND T1780  ; 3#腔体抽真空时间到达
TIMX(550) 1770 &1  ; 3#腔体抽真空NG延时
LD TR0
AND>F(333) D4156 D1230  ; #3电池真空压力表读数, 电池抽真空阀值
AND T1781  ; 3#腔电池抽真空时间到达
TIMX(550) 1771 &1  ; 3#腔电池抽真空NG延时
LD TR0
AND 12.13  ; #3电池充氦阀
AND>F(333) D4156 D1334  ; #3电池真空压力表读数, #3腔体注氦压力阀值
TIMH(015) 1772 #1  ; 3#电池注氦压力到达延时
LD TR0
AND 12.08  ; #3腔体抽气阀
TIMX(550) 1780 D1202  ; 腔体抽真空时间, 3#腔体抽真空时间到达
LD TR0
LD 12.12  ; #3电池抽气阀
OR H3.08  ; 空跑程序
ANDLD
TIMX(550) 1781 D1232  ; 电池抽真空时间, 3#腔电池抽真空时间到达
LD TR0
AND 12.13  ; #3电池充氦阀
TIMX(550) 1782 D1238  ; 注氦气时间, 3#腔注氦时间到达

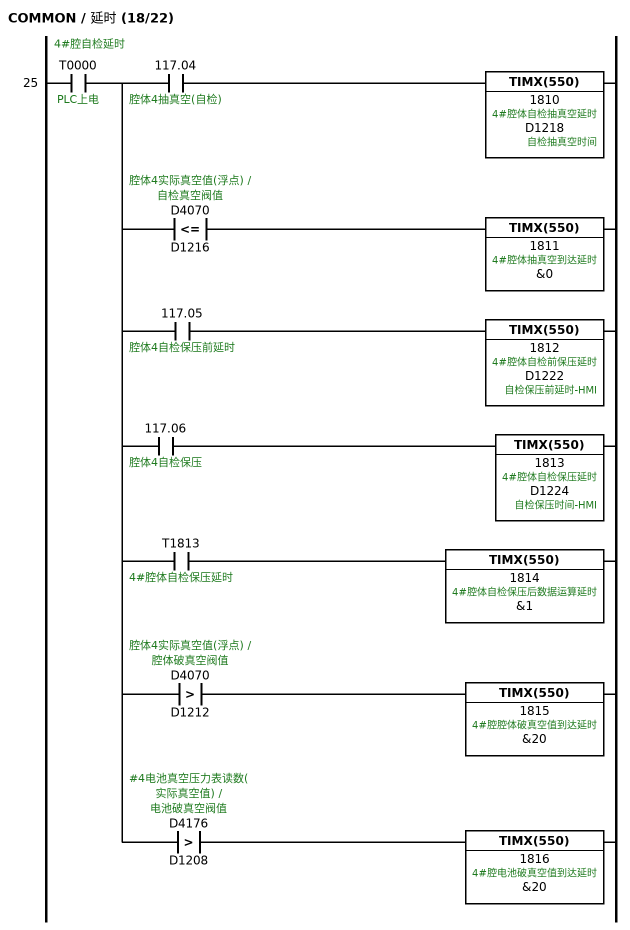
; rung 25: 4#腔自检延时
LD T0000  ; PLC上电
OUT TR0
AND 117.04  ; 腔体4抽真空(自检)
TIMX(550) 1810 D1218  ; 自检抽真空时间, 4#腔体自检抽真空延时
LD TR0
AND<=F(332) D4070 D1216  ; 腔体4实际真空值(浮点), 自检真空阀值
TIMX(550) 1811 &0  ; 4#腔体抽真空到达延时
LD TR0
AND 117.05  ; 腔体4自检保压前延时
TIMX(550) 1812 D1222  ; 自检保压前延时-HMI, 4#腔体自检前保压延时
LD TR0
AND 117.06  ; 腔体4自检保压
TIMX(550) 1813 D1224  ; 自检保压时间-HMI, 4#腔体自检保压延时
LD TR0
AND T1813  ; 4#腔体自检保压延时
TIMX(550) 1814 &1  ; 4#腔体自检保压后数据运算延时
LD TR0
AND>F(333) D4070 D1212  ; 腔体4实际真空值(浮点), 腔体破真空阀值
TIMX(550) 1815 &20  ; 4#腔腔体破真空值到达延时
LD TR0
AND>F(333) D4176 D1208  ; #4电池真空压力表读数(实际真空值), 电池破真空阀值
TIMX(550) 1816 &20  ; 4#腔电池破真空值到达延时

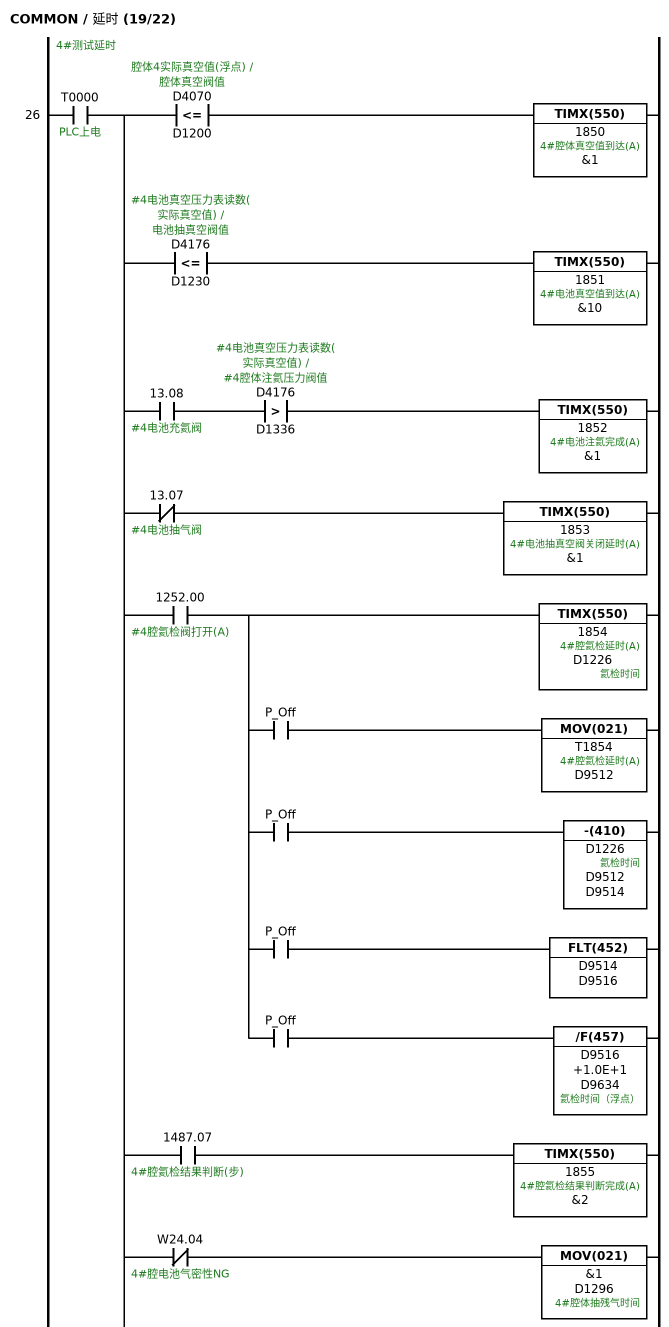

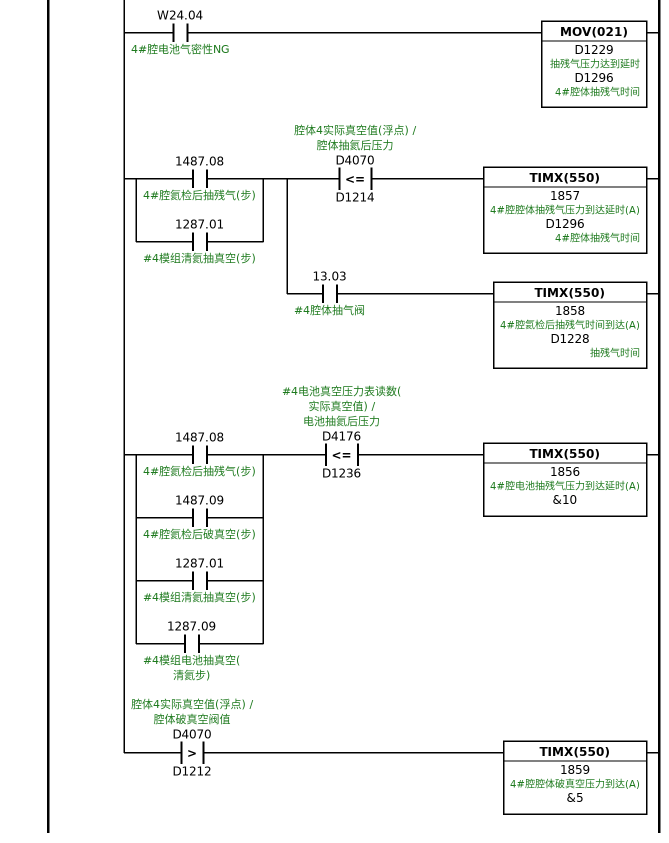
; rung 26: 4#测试延时
LD T0000  ; PLC上电
OUT TR0
AND<=F(332) D4070 D1200  ; 腔体4实际真空值(浮点), 腔体真空阀值
TIMX(550) 1850 &1  ; 4#腔体真空值到达(A)
LD TR0
AND<=F(332) D4176 D1230  ; #4电池真空压力表读数(实际真空值), 电池抽真空阀值
TIMX(550) 1851 &10  ; 4#电池真空值到达(A)
LD TR0
AND 13.08  ; #4电池充氦阀
AND>F(333) D4176 D1336  ; #4电池真空压力表读数(实际真空值), #4腔体注氦压力阀值
TIMX(550) 1852 &1  ; 4#电池注氦完成(A)
LD TR0
ANDNOT 13.07  ; #4电池抽气阀
TIMX(550) 1853 &1  ; 4#电池抽真空阀关闭延时(A)
LD TR0
AND 1252.00  ; #4腔氦检阀打开(A)
OUT TR1
TIMX(550) 1854 D1226  ; 氦检时间, 4#腔氦检延时(A)
AND P_Off
MOV(021) T1854 D9512  ; 4#腔氦检延时(A)
LD TR1
AND P_Off
-(410) D1226 D9512 D9514  ; 氦检时间
LD TR1
AND P_Off
FLT(452) D9514 D9516
LD TR1
AND P_Off
/F(457) D9516 +1.0E+1 D9634  ; 氦检时间（浮点）
LD TR0
AND 1487.07  ; 4#腔氦检结果判断(步)
TIMX(550) 1855 &2  ; 4#腔氦检结果判断完成(A)
LD TR0
ANDNOT W24.04  ; 4#腔电池气密性NG
MOV(021) &1 D1296  ; 4#腔体抽残气时间
LD TR0
AND W24.04  ; 4#腔电池气密性NG
MOV(021) D1229 D1296  ; 抽残气压力达到延时, 4#腔体抽残气时间
LD TR0
LD 1487.08  ; 4#腔氦检后抽残气(步)
OR 1287.01  ; #4模组清氦抽真空(步)
ANDLD
OUT TR1
AND<=F(332) D4070 D1214  ; 腔体4实际真空值(浮点), 腔体抽氦后压力
TIMX(550) 1857 D1296  ; 4#腔体抽残气时间, 4#腔腔体抽残气压力到达延时(A)
LD TR1
AND 13.03  ; #4腔体抽气阀
TIMX(550) 1858 D1228  ; 抽残气时间, 4#腔氦检后抽残气时间到达(A)
LD TR0
LD 1487.08  ; 4#腔氦检后抽残气(步)
OR 1487.09  ; 4#腔氦检后破真空(步)
OR 1287.01  ; #4模组清氦抽真空(步)
OR 1287.09  ; #4模组电池抽真空(清氦步)
ANDLD
AND<=F(332) D4176 D1236  ; #4电池真空压力表读数(实际真空值), 电池抽氦后压力
TIMX(550) 1856 &10  ; 4#腔电池抽残气压力到达延时(A)
LD TR0
AND>F(333) D4070 D1212  ; 腔体4实际真空值(浮点), 腔体破真空阀值
TIMX(550) 1859 &5  ; 4#腔腔体破真空压力到达(A)

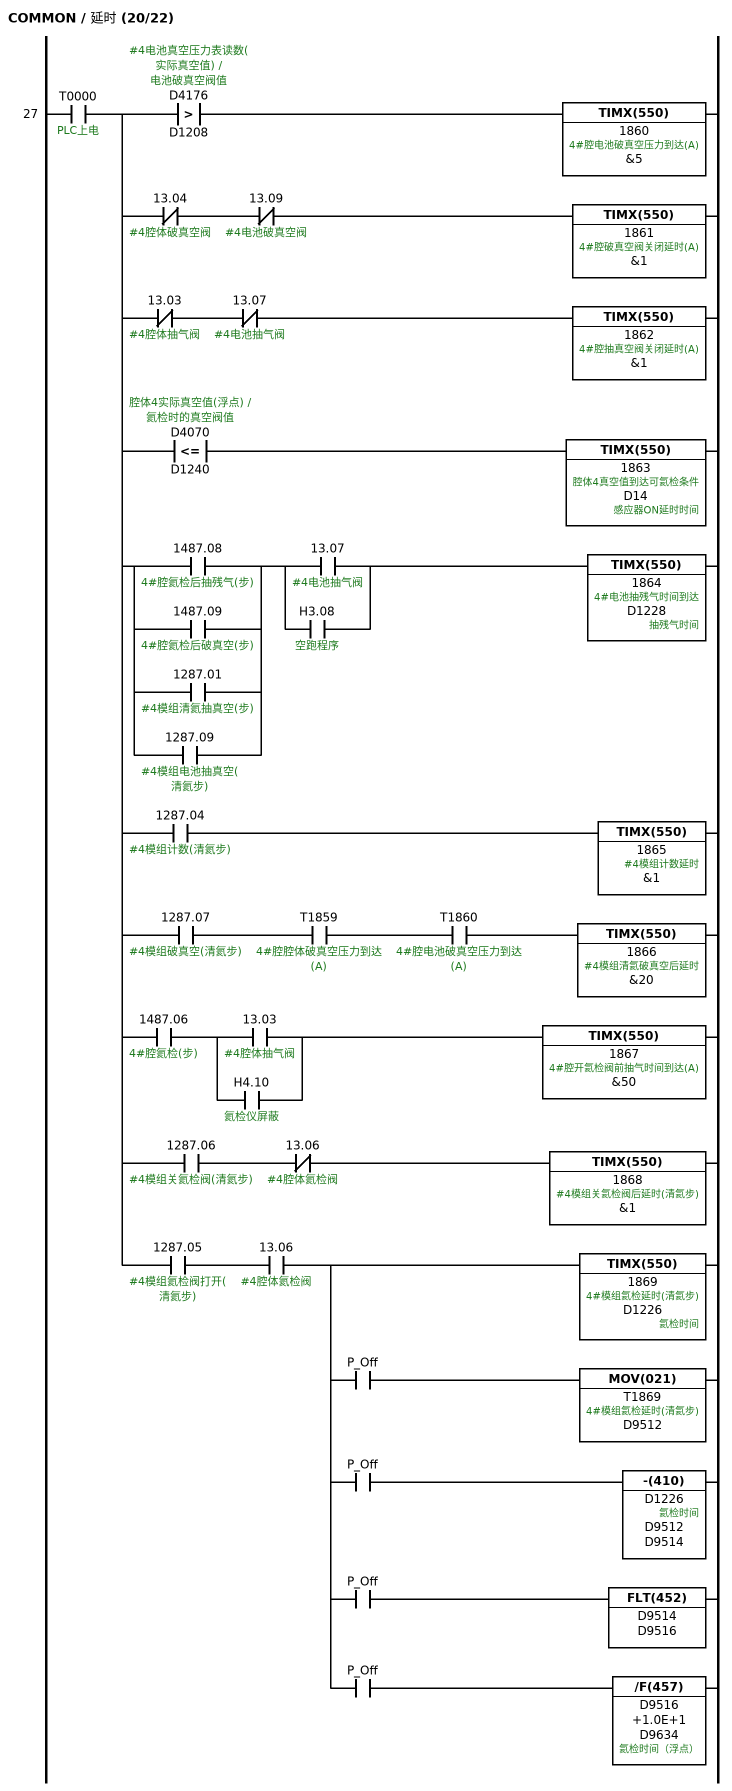
; rung 27
LD T0000  ; PLC上电
OUT TR0
AND>F(333) D4176 D1208  ; #4电池真空压力表读数(实际真空值), 电池破真空阀值
TIMX(550) 1860 &5  ; 4#腔电池破真空压力到达(A)
LD TR0
ANDNOT 13.04  ; #4腔体破真空阀
ANDNOT 13.09  ; #4电池破真空阀
TIMX(550) 1861 &1  ; 4#腔破真空阀关闭延时(A)
LD TR0
ANDNOT 13.03  ; #4腔体抽气阀
ANDNOT 13.07  ; #4电池抽气阀
TIMX(550) 1862 &1  ; 4#腔抽真空阀关闭延时(A)
LD TR0
AND<=F(332) D4070 D1240  ; 腔体4实际真空值(浮点), 氦检时的真空阀值
TIMX(550) 1863 D14  ; 感应器ON延时时间, 腔体4真空值到达可氦检条件
LD TR0
LD 1487.08  ; 4#腔氦检后抽残气(步)
OR 1487.09  ; 4#腔氦检后破真空(步)
OR 1287.01  ; #4模组清氦抽真空(步)
OR 1287.09  ; #4模组电池抽真空(清氦步)
ANDLD
LD 13.07  ; #4电池抽气阀
OR H3.08  ; 空跑程序
ANDLD
TIMX(550) 1864 D1228  ; 抽残气时间, 4#电池抽残气时间到达
LD TR0
AND 1287.04  ; #4模组计数(清氦步)
TIMX(550) 1865 &1  ; #4模组计数延时
LD TR0
AND 1287.07  ; #4模组破真空(清氦步)
AND T1859  ; 4#腔腔体破真空压力到达(A)
AND T1860  ; 4#腔电池破真空压力到达(A)
TIMX(550) 1866 &20  ; #4模组清氦破真空后延时
LD TR0
AND 1487.06  ; 4#腔氦检(步)
LD 13.03  ; #4腔体抽气阀
OR H4.10  ; 氦检仪屏蔽
ANDLD
TIMX(550) 1867 &50  ; 4#腔开氦检阀前抽气时间到达(A)
LD TR0
AND 1287.06  ; #4模组关氦检阀(清氦步)
ANDNOT 13.06  ; #4腔体氦检阀
TIMX(550) 1868 &1  ; #4模组关氦检阀后延时(清氦步)
LD TR0
AND 1287.05  ; #4模组氦检阀打开(清氦步)
AND 13.06  ; #4腔体氦检阀
OUT TR0
TIMX(550) 1869 D1226  ; 氦检时间, 4#模组氦检延时(清氦步)
AND P_Off
MOV(021) T1869 D9512  ; 4#模组氦检延时(清氦步)
LD TR0
AND P_Off
-(410) D1226 D9512 D9514  ; 氦检时间
LD TR0
AND P_Off
FLT(452) D9514 D9516
LD TR0
AND P_Off
/F(457) D9516 +1.0E+1 D9634  ; 氦检时间（浮点）

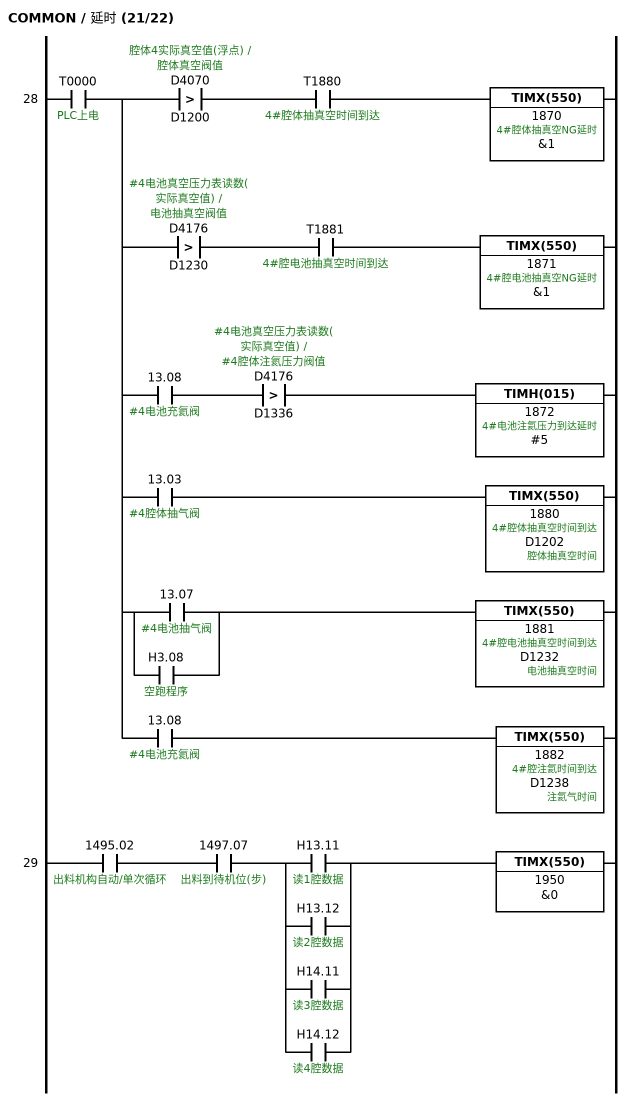
; rung 28
LD T0000  ; PLC上电
OUT TR0
AND>F(333) D4070 D1200  ; 腔体4实际真空值(浮点), 腔体真空阀值
AND T1880  ; 4#腔体抽真空时间到达
TIMX(550) 1870 &1  ; 4#腔体抽真空NG延时
LD TR0
AND>F(333) D4176 D1230  ; #4电池真空压力表读数(实际真空值), 电池抽真空阀值
AND T1881  ; 4#腔电池抽真空时间到达
TIMX(550) 1871 &1  ; 4#腔电池抽真空NG延时
LD TR0
AND 13.08  ; #4电池充氦阀
AND>F(333) D4176 D1336  ; #4电池真空压力表读数(实际真空值), #4腔体注氦压力阀值
TIMH(015) 1872 #5  ; 4#电池注氦压力到达延时
LD TR0
AND 13.03  ; #4腔体抽气阀
TIMX(550) 1880 D1202  ; 腔体抽真空时间, 4#腔体抽真空时间到达
LD TR0
LD 13.07  ; #4电池抽气阀
OR H3.08  ; 空跑程序
ANDLD
TIMX(550) 1881 D1232  ; 电池抽真空时间, 4#腔电池抽真空时间到达
LD TR0
AND 13.08  ; #4电池充氦阀
TIMX(550) 1882 D1238  ; 注氦气时间, 4#腔注氦时间到达
; rung 29
LD 1495.02  ; 出料机构自动/单次循环
AND 1497.07  ; 出料到待机位(步)
LD H13.11  ; 读1腔数据
OR H13.12  ; 读2腔数据
OR H14.11  ; 读3腔数据
OR H14.12  ; 读4腔数据
ANDLD
TIMX(550) 1950 &0

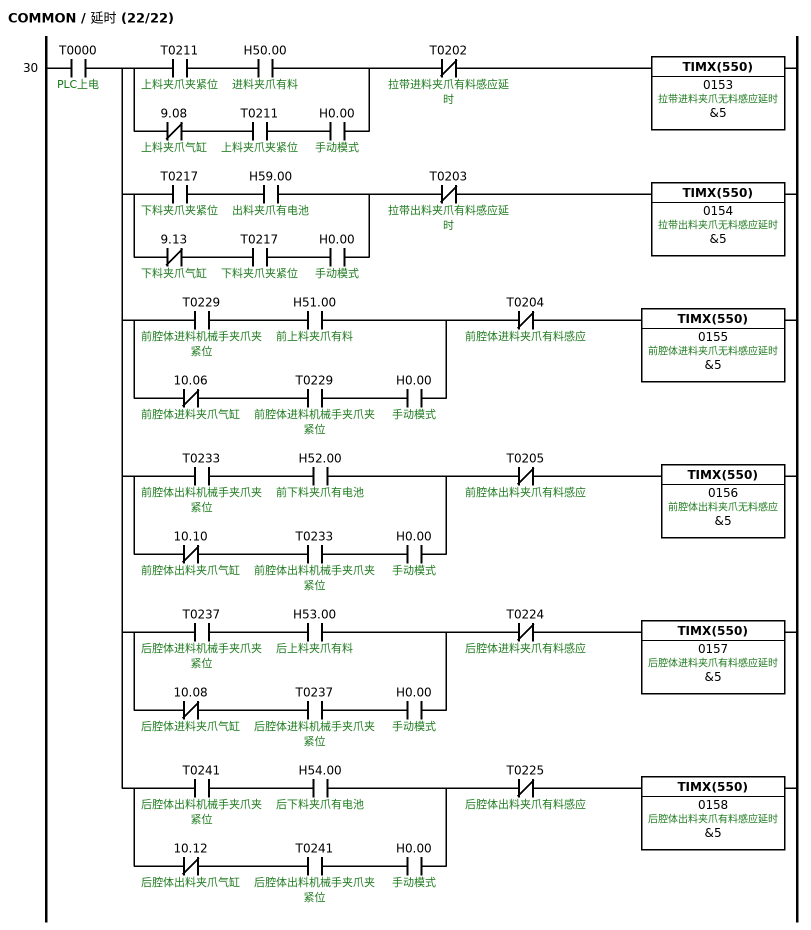
; rung 30
LD T0000  ; PLC上电
OUT TR0
LD T0211  ; 上料夹爪夹紧位
AND H50.00  ; 进料夹爪有料
LDNOT 9.08  ; 上料夹爪气缸
AND T0211  ; 上料夹爪夹紧位
AND H0.00  ; 手动模式
ORLD
ANDLD
ANDNOT T0202  ; 拉带进料夹爪有料感应延时
TIMX(550) 0153 &5  ; 拉带进料夹爪无料感应延时
LD TR0
LD T0217  ; 下料夹爪夹紧位
AND H59.00  ; 出料夹爪有电池
LDNOT 9.13  ; 下料夹爪气缸
AND T0217  ; 下料夹爪夹紧位
AND H0.00  ; 手动模式
ORLD
ANDLD
ANDNOT T0203  ; 拉带出料夹爪有料感应延时
TIMX(550) 0154 &5  ; 拉带出料夹爪无料感应延时
LD TR0
LD T0229  ; 前腔体进料机械手夹爪夹紧位
AND H51.00  ; 前上料夹爪有料
LDNOT 10.06  ; 前腔体进料夹爪气缸
AND T0229  ; 前腔体进料机械手夹爪夹紧位
AND H0.00  ; 手动模式
ORLD
ANDLD
ANDNOT T0204  ; 前腔体进料夹爪有料感应
TIMX(550) 0155 &5  ; 前腔体进料夹爪无料感应延时
LD TR0
LD T0233  ; 前腔体出料机械手夹爪夹紧位
AND H52.00  ; 前下料夹爪有电池
LDNOT 10.10  ; 前腔体出料夹爪气缸
AND T0233  ; 前腔体出料机械手夹爪夹紧位
AND H0.00  ; 手动模式
ORLD
ANDLD
ANDNOT T0205  ; 前腔体出料夹爪有料感应
TIMX(550) 0156 &5  ; 前腔体出料夹爪无料感应
LD TR0
LD T0237  ; 后腔体进料机械手夹爪夹紧位
AND H53.00  ; 后上料夹爪有料
LDNOT 10.08  ; 后腔体进料夹爪气缸
AND T0237  ; 后腔体进料机械手夹爪夹紧位
AND H0.00  ; 手动模式
ORLD
ANDLD
ANDNOT T0224  ; 后腔体进料夹爪有料感应
TIMX(550) 0157 &5  ; 后腔体进料夹爪有料感应延时
LD TR0
LD T0241  ; 后腔体出料机械手夹爪夹紧位
AND H54.00  ; 后下料夹爪有电池
LDNOT 10.12  ; 后腔体出料夹爪气缸
AND T0241  ; 后腔体出料机械手夹爪夹紧位
AND H0.00  ; 手动模式
ORLD
ANDLD
ANDNOT T0225  ; 后腔体出料夹爪有料感应
TIMX(550) 0158 &5  ; 后腔体出料夹爪有料感应延时

### Section 感应器延时

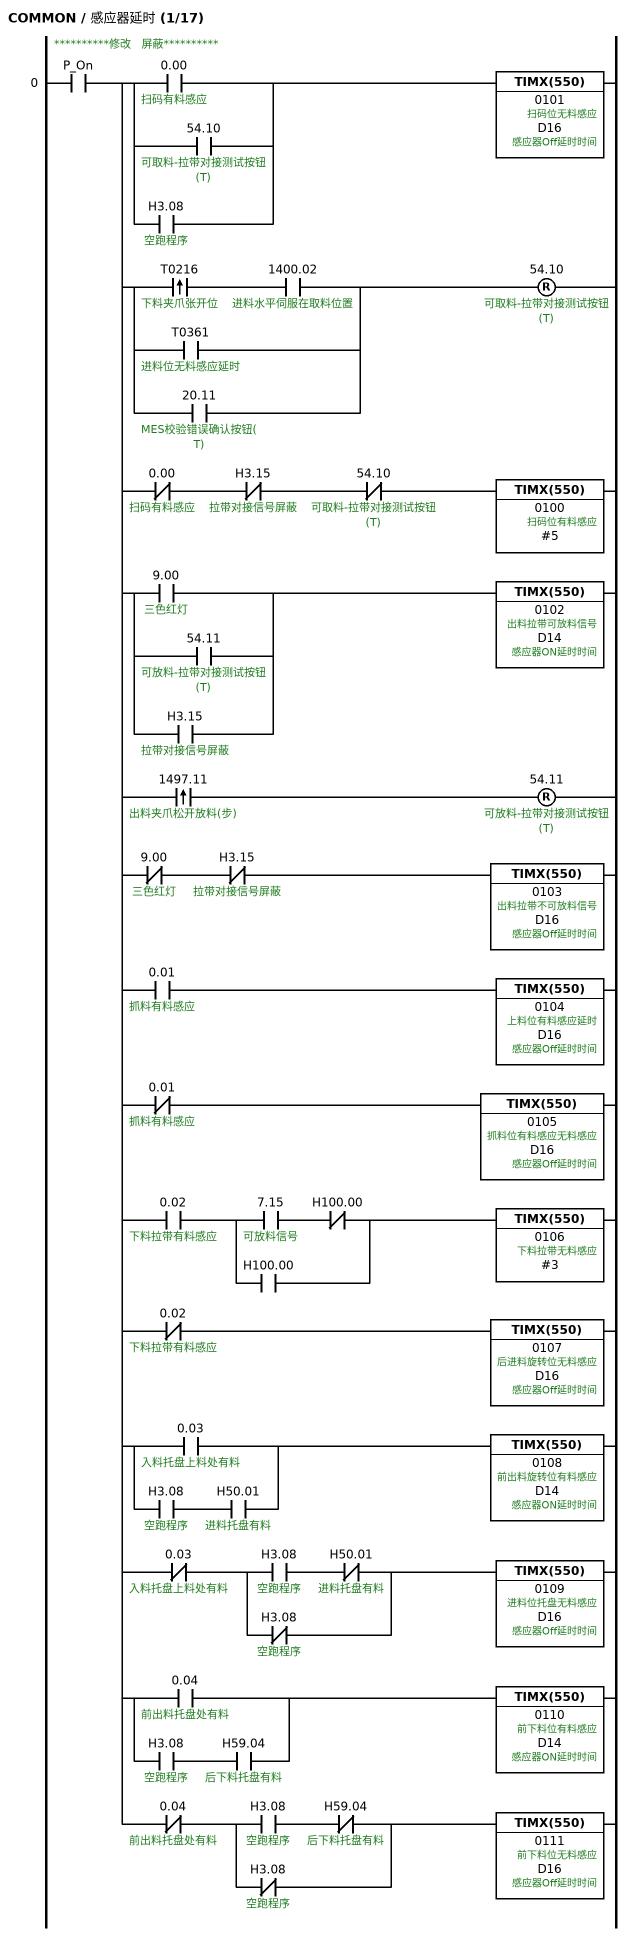
; rung 0: **********修改   屏蔽**********
LD P_On
OUT TR0
LD 0.00  ; 扫码有料感应
OR 54.10  ; 可取料-拉带对接测试按钮(T)
OR H3.08  ; 空跑程序
ANDLD
TIMX(550) 0101 D16  ; 感应器Off延时时间, 扫码位无料感应
LD TR0
@LD T0216  ; 下料夹爪张开位
AND 1400.02  ; 进料水平伺服在取料位置
OR T0361  ; 进料位无料感应延时
OR 20.11  ; MES校验错误确认按钮(T)
ANDLD
RSET 54.10  ; 可取料-拉带对接测试按钮(T)
LD TR0
ANDNOT 0.00  ; 扫码有料感应
ANDNOT H3.15  ; 拉带对接信号屏蔽
ANDNOT 54.10  ; 可取料-拉带对接测试按钮(T)
TIMX(550) 0100 #5  ; 扫码位有料感应
LD TR0
LD 9.00  ; 三色红灯
OR 54.11  ; 可放料-拉带对接测试按钮(T)
OR H3.15  ; 拉带对接信号屏蔽
ANDLD
TIMX(550) 0102 D14  ; 感应器ON延时时间, 出料拉带可放料信号
LD TR0
@AND 1497.11  ; 出料夹爪松开放料(步)
RSET 54.11  ; 可放料-拉带对接测试按钮(T)
LD TR0
ANDNOT 9.00  ; 三色红灯
ANDNOT H3.15  ; 拉带对接信号屏蔽
TIMX(550) 0103 D16  ; 感应器Off延时时间, 出料拉带不可放料信号
LD TR0
AND 0.01  ; 抓料有料感应
TIMX(550) 0104 D16  ; 感应器Off延时时间, 上料位有料感应延时
LD TR0
ANDNOT 0.01  ; 抓料有料感应
TIMX(550) 0105 D16  ; 感应器Off延时时间, 抓料位有料感应无料感应
LD TR0
AND 0.02  ; 下料拉带有料感应
LD 7.15  ; 可放料信号
ANDNOT H100.00
OR H100.00
ANDLD
TIMX(550) 0106 #3  ; 下料拉带无料感应
LD TR0
ANDNOT 0.02  ; 下料拉带有料感应
TIMX(550) 0107 D16  ; 感应器Off延时时间, 后进料旋转位无料感应
LD TR0
LD 0.03  ; 入料托盘上料处有料
LD H3.08  ; 空跑程序
AND H50.01  ; 进料托盘有料
ORLD
ANDLD
TIMX(550) 0108 D14  ; 感应器ON延时时间, 前出料旋转位有料感应
LD TR0
ANDNOT 0.03  ; 入料托盘上料处有料
LD H3.08  ; 空跑程序
ANDNOT H50.01  ; 进料托盘有料
ORNOT H3.08  ; 空跑程序
ANDLD
TIMX(550) 0109 D16  ; 感应器Off延时时间, 进料位托盘无料感应
LD TR0
LD 0.04  ; 前出料托盘处有料
LD H3.08  ; 空跑程序
AND H59.04  ; 后下料托盘有料
ORLD
ANDLD
TIMX(550) 0110 D14  ; 感应器ON延时时间, 前下料位有料感应
LD TR0
ANDNOT 0.04  ; 前出料托盘处有料
LD H3.08  ; 空跑程序
ANDNOT H59.04  ; 后下料托盘有料
ORNOT H3.08  ; 空跑程序
ANDLD
TIMX(550) 0111 D16  ; 感应器Off延时时间, 前下料位无料感应

